# EPICS autosave request: iocBoot/scanPv.req
$(P):SCANPV1:INC
$(P):SCANPV1:SPEED
$(P):SCANPV1:START
$(P):SCANPV1:STOP
$(P):SCANPV1:NSTEPS
$(P):SCANPV1:DESC
$(P):SCANPV1:OFFSET
$(P):SCANPV1:SETTLETIME
$(P):SCANPV1:PVNAME
$(P):SCANPV1:PVTYPE
$(P):SCANPV1:DELTA
$(P):SCANPV1:PRE_START
$(P):SCANPV1:PRE_STOP
$(P):SCANPV1:PRE_NSTEPS
$(P):SCANPV1:PRE_INC
$(P):SCANPV1:RANDSCAN
$(P):SCANPV1:RAND_VALS
$(P):SCANPV1:RBVNAME

$(P):SCANPV2:INC
$(P):SCANPV2:SPEED
$(P):SCANPV2:START
$(P):SCANPV2:STOP
$(P):SCANPV2:NSTEPS
$(P):SCANPV2:DESC
$(P):SCANPV2:OFFSET
$(P):SCANPV2:SETTLETIME
$(P):SCANPV2:PVNAME
$(P):SCANPV2:PVTYPE
$(P):SCANPV2:DELTA
$(P):SCANPV2:PRE_START
$(P):SCANPV2:PRE_STOP
$(P):SCANPV2:PRE_NSTEPS
$(P):SCANPV2:PRE_INC
$(P):SCANPV2:RANDSCAN
$(P):SCANPV2:RAND_VALS
$(P):SCANPV2:RBVNAME

$(P):SCANPV3:INC
$(P):SCANPV3:SPEED
$(P):SCANPV3:START
$(P):SCANPV3:STOP
$(P):SCANPV3:NSTEPS
$(P):SCANPV3:DESC
$(P):SCANPV3:OFFSET
$(P):SCANPV3:SETTLETIME
$(P):SCANPV3:PVNAME
$(P):SCANPV3:PVTYPE
$(P):SCANPV3:DELTA
$(P):SCANPV3:PRE_START
$(P):SCANPV3:PRE_STOP
$(P):SCANPV3:PRE_NSTEPS
$(P):SCANPV3:PRE_INC
$(P):SCANPV3:RANDSCAN
$(P):SCANPV3:RAND_VALS
$(P):SCANPV3:RBVNAME

$(P):SCANPV4:INC
$(P):SCANPV4:SPEED
$(P):SCANPV4:START
$(P):SCANPV4:STOP
$(P):SCANPV4:NSTEPS
$(P):SCANPV4:DESC
$(P):SCANPV4:OFFSET
$(P):SCANPV4:SETTLETIME
$(P):SCANPV4:PVNAME
$(P):SCANPV4:PVTYPE
$(P):SCANPV4:DELTA
$(P):SCANPV4:PRE_START
$(P):SCANPV4:PRE_STOP
$(P):SCANPV4:PRE_NSTEPS
$(P):SCANPV4:PRE_INC
$(P):SCANPV4:RANDSCAN
$(P):SCANPV4:RAND_VALS
$(P):SCANPV4:RBVNAME

$(P):SCANPV5:INC
$(P):SCANPV5:SPEED
$(P):SCANPV5:START
$(P):SCANPV5:STOP
$(P):SCANPV5:NSTEPS
$(P):SCANPV5:DESC
$(P):SCANPV5:OFFSET
$(P):SCANPV5:SETTLETIME
$(P):SCANPV5:PVNAME
$(P):SCANPV5:PVTYPE
$(P):SCANPV5:DELTA
$(P):SCANPV5:PRE_START
$(P):SCANPV5:PRE_STOP
$(P):SCANPV5:PRE_NSTEPS
$(P):SCANPV5:PRE_INC
$(P):SCANPV5:RANDSCAN
$(P):SCANPV5:RAND_VALS
$(P):SCANPV5:RBVNAME

$(P):SCANPV6:INC
$(P):SCANPV6:SPEED
$(P):SCANPV6:START
$(P):SCANPV6:STOP
$(P):SCANPV6:NSTEPS
$(P):SCANPV6:DESC
$(P):SCANPV6:OFFSET
$(P):SCANPV6:SETTLETIME
$(P):SCANPV6:PVNAME
$(P):SCANPV6:PVTYPE
$(P):SCANPV6:DELTA
$(P):SCANPV6:PRE_START
$(P):SCANPV6:PRE_STOP
$(P):SCANPV6:PRE_NSTEPS
$(P):SCANPV6:PRE_INC
$(P):SCANPV6:RANDSCAN
$(P):SCANPV6:RAND_VALS
$(P):SCANPV6:RBVNAME

$(P):SCANPV7:INC
$(P):SCANPV7:SPEED
$(P):SCANPV7:START
$(P):SCANPV7:STOP
$(P):SCANPV7:NSTEPS
$(P):SCANPV7:DESC
$(P):SCANPV7:OFFSET
$(P):SCANPV7:SETTLETIME
$(P):SCANPV7:PVNAME
$(P):SCANPV7:PVTYPE
$(P):SCANPV7:DELTA
$(P):SCANPV7:PRE_START
$(P):SCANPV7:PRE_STOP
$(P):SCANPV7:PRE_NSTEPS
$(P):SCANPV7:PRE_INC
$(P):SCANPV7:RANDSCAN
$(P):SCANPV7:RAND_VALS
$(P):SCANPV7:RBVNAME

$(P):SCANPV8:INC
$(P):SCANPV8:SPEED
$(P):SCANPV8:START
$(P):SCANPV8:STOP
$(P):SCANPV8:NSTEPS
$(P):SCANPV8:DESC
$(P):SCANPV8:OFFSET
$(P):SCANPV8:SETTLETIME
$(P):SCANPV8:PVNAME
$(P):SCANPV8:PVTYPE
$(P):SCANPV8:DELTA
$(P):SCANPV8:PRE_START
$(P):SCANPV8:PRE_STOP
$(P):SCANPV8:PRE_NSTEPS
$(P):SCANPV8:PRE_INC
$(P):SCANPV8:RANDSCAN
$(P):SCANPV8:RAND_VALS
$(P):SCANPV8:RBVNAME

$(P):SCANPV9:INC
$(P):SCANPV9:SPEED
$(P):SCANPV9:START
$(P):SCANPV9:STOP
$(P):SCANPV9:NSTEPS
$(P):SCANPV9:DESC
$(P):SCANPV9:OFFSET
$(P):SCANPV9:SETTLETIME
$(P):SCANPV9:PVNAME
$(P):SCANPV9:PVTYPE
$(P):SCANPV9:DELTA
$(P):SCANPV9:PRE_START
$(P):SCANPV9:PRE_STOP
$(P):SCANPV9:PRE_NSTEPS
$(P):SCANPV9:PRE_INC
$(P):SCANPV9:RANDSCAN
$(P):SCANPV9:RAND_VALS
$(P):SCANPV9:RBVNAME

$(P):SCANPV10:INC
$(P):SCANPV10:SPEED
$(P):SCANPV10:START
$(P):SCANPV10:STOP
$(P):SCANPV10:NSTEPS
$(P):SCANPV10:DESC
$(P):SCANPV10:OFFSET
$(P):SCANPV10:SETTLETIME
$(P):SCANPV10:PVNAME
$(P):SCANPV10:PVTYPE
$(P):SCANPV10:DELTA
$(P):SCANPV10:PRE_START
$(P):SCANPV10:PRE_STOP
$(P):SCANPV10:PRE_NSTEPS
$(P):SCANPV10:PRE_INC
$(P):SCANPV10:RANDSCAN
$(P):SCANPV10:RAND_VALS
$(P):SCANPV10:RBVNAME
